FUNCTION_BLOCK BatteryActor (* Actor for sending data to the BatteryActor plugin controller in Polysun. *)
  (* Standard: 61499-2 *)
  (* Version 1.0, 2017-07-21, Marc Jakobi, HTW Berlin *)
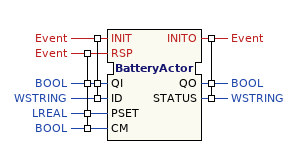
  EVENT_INPUT
    INIT WITH QI, ID; (* Service Initialization *)
    RSP WITH PSET, CM, QI; (* Service Response *)
  END_EVENT
  EVENT_OUTPUT
    INITO WITH QO, STATUS; (* Initialization Confirm *)
  END_EVENT
  VAR_INPUT
    QI : BOOL; (* Input event qualifier *)
    ID : WSTRING; (* Connection identifier *)
    PSET : LREAL; (* Set charging power in W *)
    CM : BOOL; (* Control mode *)
  END_VAR
  VAR_OUTPUT
    QO : BOOL; (* Output event qualifier *)
    STATUS : WSTRING; (* Service status *)
  END_VAR
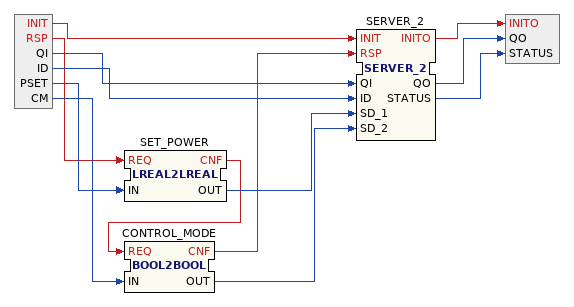
  FBS
    SERVER_2 : SERVER_2;
    SET_POWER : LREAL2LREAL;
    CONTROL_MODE : BOOL2BOOL;
  END_FBS
  EVENT_CONNECTIONS
    INIT TO SERVER_2.INIT;
    SERVER_2.INITO TO INITO;
    RSP TO SET_POWER.REQ;
    SET_POWER.CNF TO CONTROL_MODE.REQ;
    CONTROL_MODE.CNF TO SERVER_2.RSP;
  END_CONNECTIONS
  DATA_CONNECTIONS
    QI TO SERVER_2.QI;
    ID TO SERVER_2.ID;
    SERVER_2.QO TO QO;
    SERVER_2.STATUS TO STATUS;
    PSET TO SET_POWER.IN;
    SET_POWER.OUT TO SERVER_2.SD_1;
    CM TO CONTROL_MODE.IN;
    CONTROL_MODE.OUT TO SERVER_2.SD_2;
  END_CONNECTIONS
END_FUNCTION_BLOCK
